Staubli VAL3: recvMsgHeader.pgx

public program recvMsgHeader(sio& x_sSocket (dimensions=1), num& x_nConnFlag (dimensions=1), RosSimpleMsg& x_msg (dimensions=1), num& x_nMsgRecvState (dimensions=1))
  local bool l_bFlag
begin
  // Copyright (c) 2016, Ocado Technology - Robotics Research Team
  // Copyright (c) 2021, Institute for Factory Automation and Production Systems (FAPS)
  //
  // Licensed under the Apache License, Version 2.0 (the "License");
  // you may not use this file except in compliance with the License.
  // You may obtain a copy of the License at
  //
  //     http://www.apache.org/licenses/LICENSE-2.0
  //
  // Unless required by applicable law or agreed to in writing, software
  // distributed under the License is distributed on an "AS IS" BASIS,
  // WITHOUT WARRANTIES OR CONDITIONS OF ANY KIND, either express or implied.
  // See the License for the specific language governing permissions and
  // limitations under the License.



  // attempt to receive message prefix and header
  call recvData(x_sSocket,x_msg.prefix.nData,x_nConnFlag,l_bFlag)
  if (l_bFlag==true)
    call recvData(x_sSocket,x_msg.header.nData,x_nConnFlag,l_bFlag)
  endIf

  if (l_bFlag == true)
    // move on to state 1: decode header
    x_nMsgRecvState = MsgRecvState.DECODE_HEADER
  else
    // error: reset state to 0: receive header
    x_nMsgRecvState = MsgRecvState.RECEIVE_HEADER
  endIf
end
